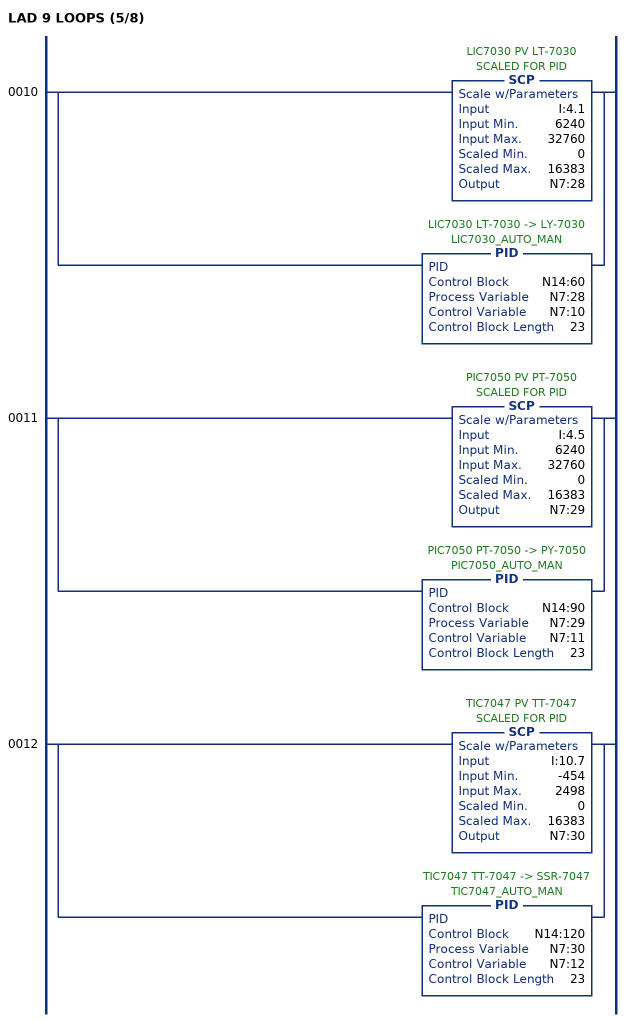
% Rung: 10 %
SOR BST SCP I:4.1 6240 32760 0 16383 N7:28 NXB PID N14:60 N7:28 N7:10 23 BND EOR
%   I:4.1  LT_7030  "LT-7030 ANALOG IN" %
%   N7:28  "LIC7030 PV LT-7030 SCALED FOR PID" %
%   N14:60  LIC7030_AUTO_MAN  "LIC7030 LT-7030 -> LY-7030" %
%   N7:10  "LY-7030 PID OP" %
% Rung: 11 %
SOR BST SCP I:4.5 6240 32760 0 16383 N7:29 NXB PID N14:90 N7:29 N7:11 23 BND EOR
%   I:4.5  PT_7050  "PT-7050 ANALOG IN" %
%   N7:29  "PIC7050 PV PT-7050 SCALED FOR PID" %
%   N14:90  PIC7050_AUTO_MAN  "PIC7050 PT-7050 -> PY-7050" %
%   N7:11  "PY-7050 PID OP" %
% Rung: 12 %
SOR BST SCP I:10.7 -454 2498 0 16383 N7:30 NXB PID N14:120 N7:30 N7:12 23 BND EOR
%   I:10.7  TT_7047  "TT-7047 ANALOG IN" %
%   N7:30  "TIC7047 PV TT-7047 SCALED FOR PID" %
%   N14:120  TIC7047_AUTO_MAN  "TIC7047 TT-7047 -> SSR-7047" %
%   N7:12  "SSR-7047 PID OP" %

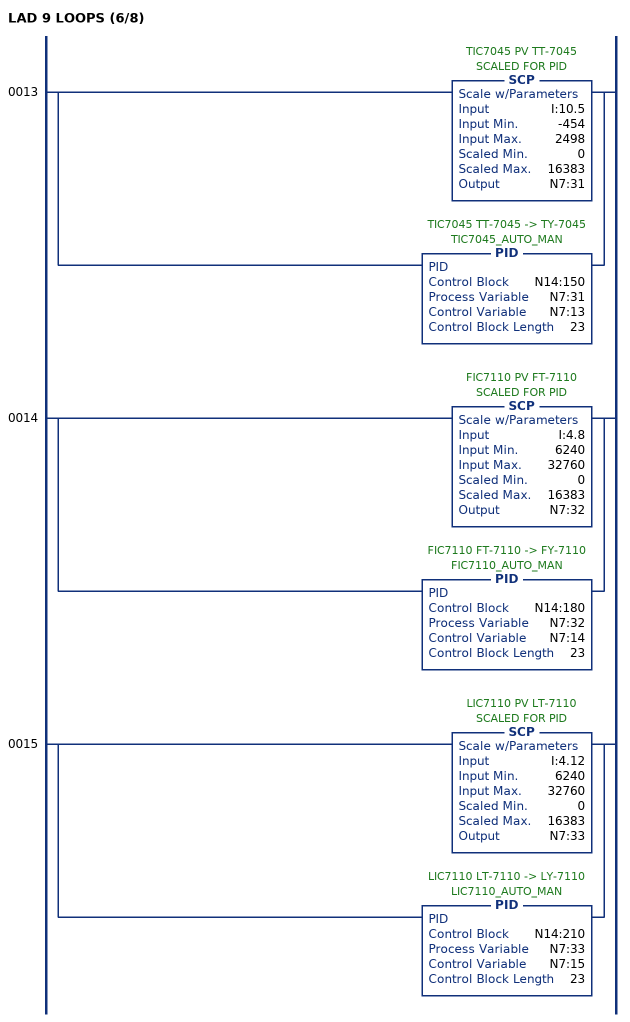
% Rung: 13 %
SOR BST SCP I:10.5 -454 2498 0 16383 N7:31 NXB PID N14:150 N7:31 N7:13 23 BND EOR
%   I:10.5  TT_7045  "TT-7045 ANALOG IN" %
%   N7:31  "TIC7045 PV TT-7045 SCALED FOR PID" %
%   N14:150  TIC7045_AUTO_MAN  "TIC7045 TT-7045 -> TY-7045" %
%   N7:13  "TY-7045 PID OP" %
% Rung: 14 %
SOR BST SCP I:4.8 6240 32760 0 16383 N7:32 NXB PID N14:180 N7:32 N7:14 23 BND EOR
%   I:4.8  FT_7110  "FT-7110 ANALOG IN" %
%   N7:32  "FIC7110 PV FT-7110 SCALED FOR PID" %
%   N14:180  FIC7110_AUTO_MAN  "FIC7110 FT-7110 -> FY-7110" %
%   N7:14  "FY-7110 PID OP" %
% Rung: 15 %
SOR BST SCP I:4.12 6240 32760 0 16383 N7:33 NXB PID N14:210 N7:33 N7:15 23 BND EOR
%   I:4.12  LT_7110  "LT-7110 ANALOG IN" %
%   N7:33  "LIC7110 PV LT-7110 SCALED FOR PID" %
%   N14:210  LIC7110_AUTO_MAN  "LIC7110 LT-7110 -> LY-7110" %
%   N7:15  "LY-7110 PID OP" %

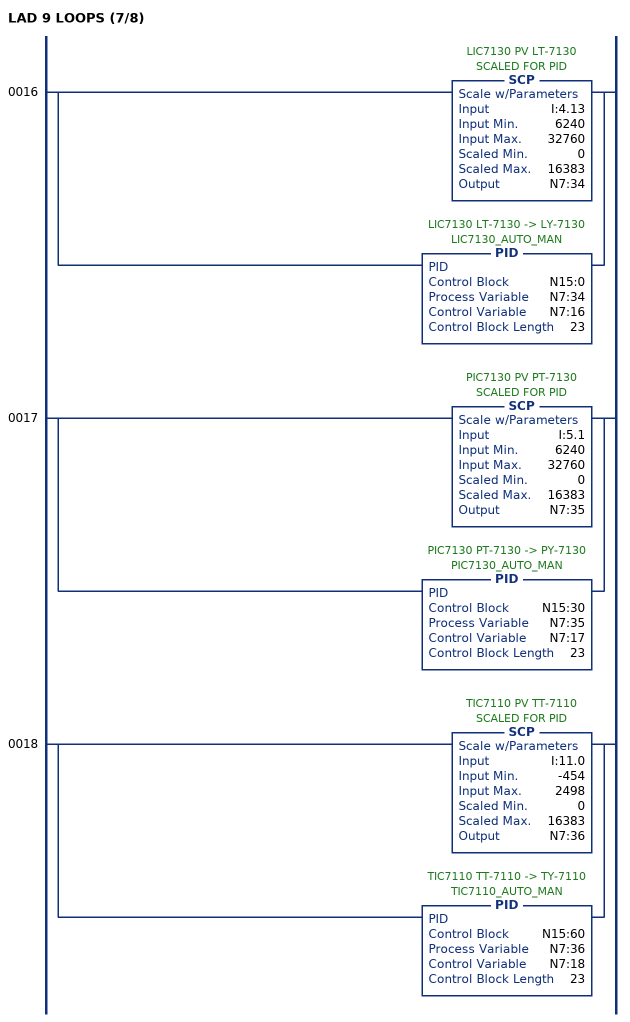
% Rung: 16 %
SOR BST SCP I:4.13 6240 32760 0 16383 N7:34 NXB PID N15:0 N7:34 N7:16 23 BND EOR
%   I:4.13  LT_7130  "LT-7130 ANALOG IN" %
%   N7:34  "LIC7130 PV LT-7130 SCALED FOR PID" %
%   N15:0  LIC7130_AUTO_MAN  "LIC7130 LT-7130 -> LY-7130" %
%   N7:16  "LY-7130 PID OP" %
% Rung: 17 %
SOR BST SCP I:5.1 6240 32760 0 16383 N7:35 NXB PID N15:30 N7:35 N7:17 23 BND EOR
%   I:5.1  PT_7130  "PT-7130 ANALOG IN" %
%   N7:35  "PIC7130 PV PT-7130 SCALED FOR PID" %
%   N15:30  PIC7130_AUTO_MAN  "PIC7130 PT-7130 -> PY-7130" %
%   N7:17  "PY-7130 PID OP" %
% Rung: 18 %
SOR BST SCP I:11.0 -454 2498 0 16383 N7:36 NXB PID N15:60 N7:36 N7:18 23 BND EOR
%   I:11.0  TT_7110  "TT-7110 ANALOG IN" %
%   N7:36  "TIC7110 PV TT-7110 SCALED FOR PID" %
%   N15:60  TIC7110_AUTO_MAN  "TIC7110 TT-7110 -> TY-7110" %
%   N7:18  "TY-7110 PID OP" %

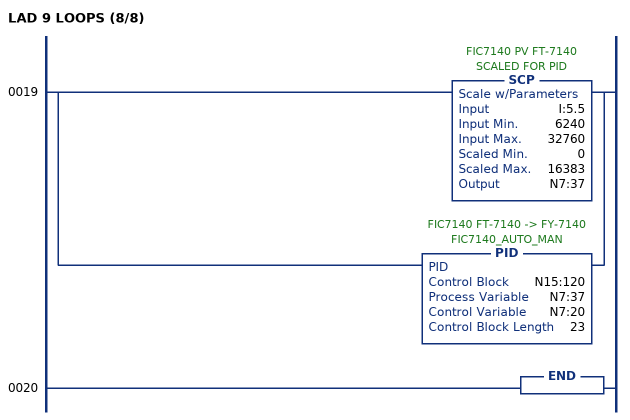
% Rung: 19 %
SOR BST SCP I:5.5 6240 32760 0 16383 N7:37 NXB PID N15:120 N7:37 N7:20 23 BND EOR
%   I:5.5  FT_7140  "FT-7140 ANALOG IN" %
%   N7:37  "FIC7140 PV FT-7140 SCALED FOR PID" %
%   N15:120  FIC7140_AUTO_MAN  "FIC7140 FT-7140 -> FY-7140" %
%   N7:20  "FY-7140 PID OP" %
% Rung: 20 %
SOR END EOR

LADDER 10 "CONTROL"
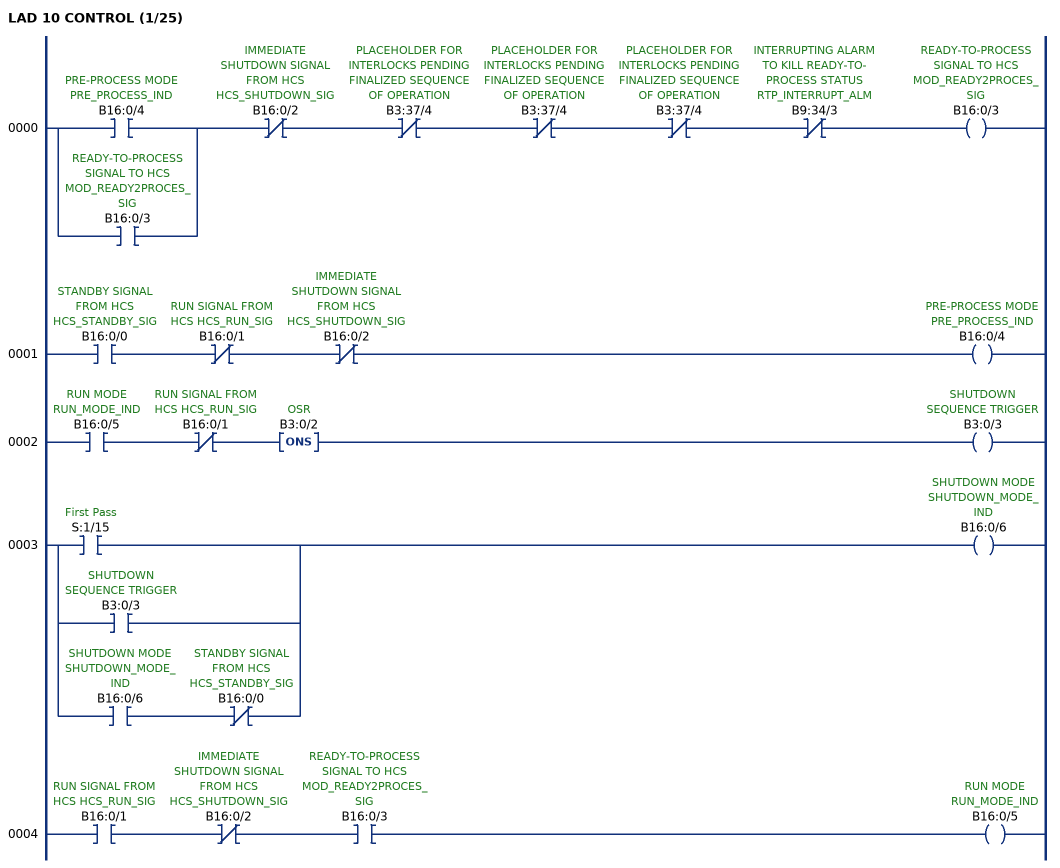
% Rung: 0 %
SOR BST XIC B16:0/4 NXB XIC B16:0/3 BND XIO B16:0/2 XIO B3:37/4 XIO B3:37/4 XIO B3:37/4 XIO B9:34/3 OTE B16:0/3 EOR
%   B16:0/4  PRE_PROCESS_IND  "PRE-PROCESS MODE" %
%   B16:0/3  MOD_READY2PROCES_SIG  "READY-TO-PROCESS SIGNAL TO HCS" %
%   B16:0/2  HCS_SHUTDOWN_SIG  "IMMEDIATE SHUTDOWN SIGNAL FROM HCS" %
%   B3:37/4  "PLACEHOLDER FOR INTERLOCKS PENDING FINALIZED SEQUENCE OF OPERATION" %
%   B9:34/3  RTP_INTERRUPT_ALM  "INTERRUPTING ALARM TO KILL READY-TO-PROCESS STATUS" %
% Rung: 1 %
SOR XIC B16:0/0 XIO B16:0/1 XIO B16:0/2 OTE B16:0/4 EOR
%   B16:0/0  HCS_STANDBY_SIG  "STANDBY SIGNAL FROM HCS" %
%   B16:0/1  HCS_RUN_SIG  "RUN SIGNAL FROM HCS" %
%   B16:0/2  HCS_SHUTDOWN_SIG  "IMMEDIATE SHUTDOWN SIGNAL FROM HCS" %
%   B16:0/4  PRE_PROCESS_IND  "PRE-PROCESS MODE" %
% Rung: 2 %
SOR XIC B16:0/5 XIO B16:0/1 OSR B3:0/2 OTE B3:0/3 EOR
%   B16:0/5  RUN_MODE_IND  "RUN MODE" %
%   B16:0/1  HCS_RUN_SIG  "RUN SIGNAL FROM HCS" %
%   B3:0/2  "OSR" %
%   B3:0/3  "SHUTDOWN SEQUENCE TRIGGER" %
% Rung: 3 %
SOR BST XIC S:1/15 NXB XIC B3:0/3 NXB XIC B16:0/6 XIO B16:0/0 BND OTE B16:0/6 EOR
%   S:1/15  "First Pass" %
%   B3:0/3  "SHUTDOWN SEQUENCE TRIGGER" %
%   B16:0/6  SHUTDOWN_MODE_IND  "SHUTDOWN MODE" %
%   B16:0/0  HCS_STANDBY_SIG  "STANDBY SIGNAL FROM HCS" %
% Rung: 4 %
SOR XIC B16:0/1 XIO B16:0/2 XIC B16:0/3 OTE B16:0/5 EOR
%   B16:0/1  HCS_RUN_SIG  "RUN SIGNAL FROM HCS" %
%   B16:0/2  HCS_SHUTDOWN_SIG  "IMMEDIATE SHUTDOWN SIGNAL FROM HCS" %
%   B16:0/3  MOD_READY2PROCES_SIG  "READY-TO-PROCESS SIGNAL TO HCS" %
%   B16:0/5  RUN_MODE_IND  "RUN MODE" %

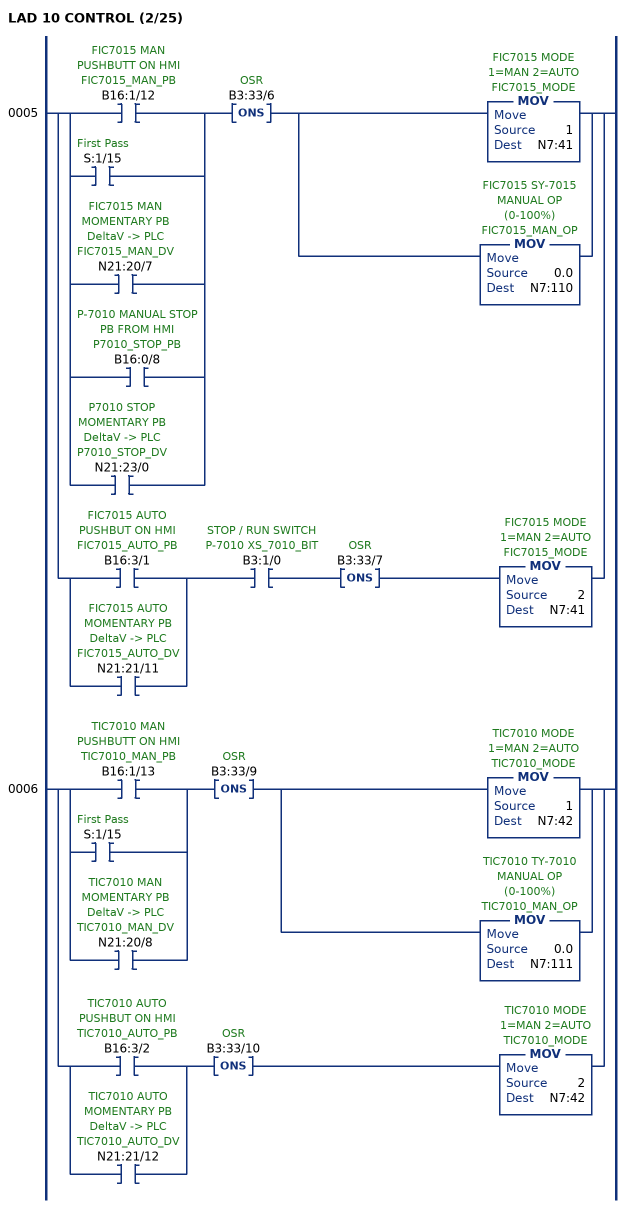
% Rung: 5 %
SOR BST BST XIC B16:1/12 NXB XIC S:1/15 NXB XIC N21:20/7 NXB XIC B16:0/8 NXB XIC N21:23/0 BND OSR B3:33/6 BST MOV 1 N7:41 NXB MOV 0.0 N7:110 BND NXB BST XIC B16:3/1 NXB XIC N21:21/11 BND XIC B3:1/0 OSR B3:33/7 MOV 2 N7:41 BND EOR
%   B16:1/12  FIC7015_MAN_PB  "FIC7015 MAN PUSHBUTT ON HMI" %
%   S:1/15  "First Pass" %
%   N21:20/7  FIC7015_MAN_DV  "FIC7015 MAN MOMENTARY PB DeltaV -> PLC" %
%   B16:0/8  P7010_STOP_PB  "P-7010 MANUAL STOP PB FROM HMI" %
%   N21:23/0  P7010_STOP_DV  "P7010 STOP MOMENTARY PB DeltaV -> PLC" %
%   B3:33/6  "OSR" %
%   N7:41  FIC7015_MODE  "FIC7015 MODE 1=MAN 2=AUTO" %
%   N7:110  FIC7015_MAN_OP  "FIC7015 SY-7015 MANUAL OP (0-100%)" %
%   B16:3/1  FIC7015_AUTO_PB  "FIC7015 AUTO PUSHBUT ON HMI" %
%   N21:21/11  FIC7015_AUTO_DV  "FIC7015 AUTO MOMENTARY PB DeltaV -> PLC" %
%   B3:1/0  XS_7010_BIT  "STOP / RUN SWITCH P-7010" %
%   B3:33/7  "OSR" %
% Rung: 6 %
SOR BST BST XIC B16:1/13 NXB XIC S:1/15 NXB XIC N21:20/8 BND OSR B3:33/9 BST MOV 1 N7:42 NXB MOV 0.0 N7:111 BND NXB BST XIC B16:3/2 NXB XIC N21:21/12 BND OSR B3:33/10 MOV 2 N7:42 BND EOR
%   B16:1/13  TIC7010_MAN_PB  "TIC7010 MAN PUSHBUTT ON HMI" %
%   S:1/15  "First Pass" %
%   N21:20/8  TIC7010_MAN_DV  "TIC7010 MAN MOMENTARY PB DeltaV -> PLC" %
%   B3:33/9  "OSR" %
%   N7:42  TIC7010_MODE  "TIC7010 MODE 1=MAN 2=AUTO" %
%   N7:111  TIC7010_MAN_OP  "TIC7010 TY-7010 MANUAL OP (0-100%)" %
%   B16:3/2  TIC7010_AUTO_PB  "TIC7010 AUTO PUSHBUT ON HMI" %
%   N21:21/12  TIC7010_AUTO_DV  "TIC7010 AUTO MOMENTARY PB DeltaV -> PLC" %
%   B3:33/10  "OSR" %

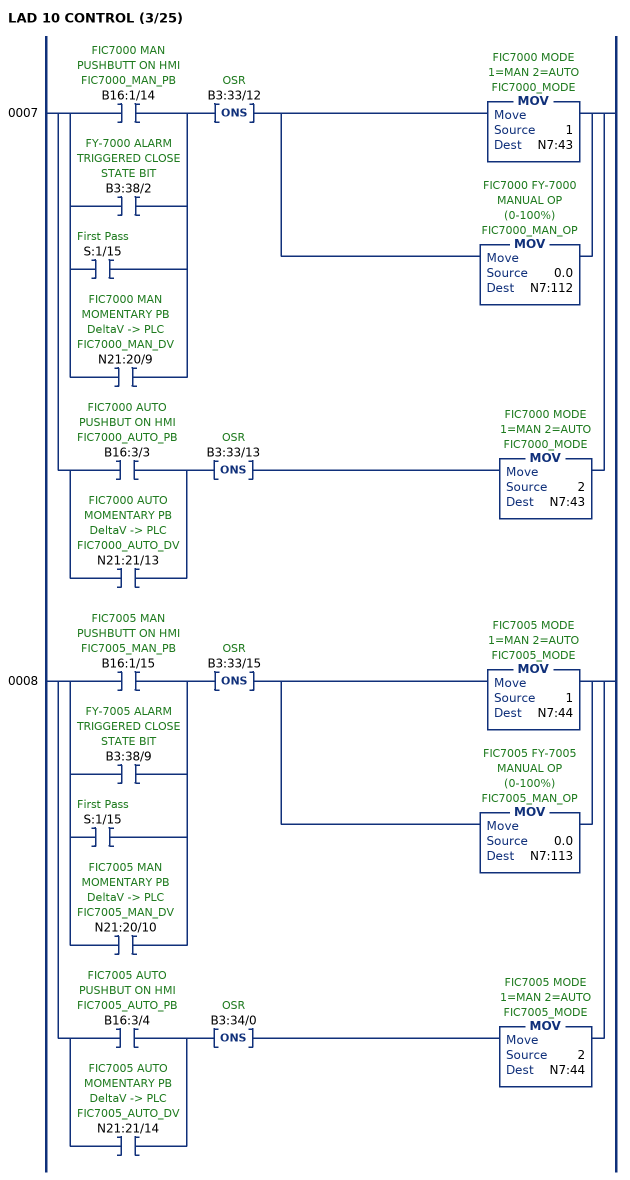
% Rung: 7 %
SOR BST BST XIC B16:1/14 NXB XIC B3:38/2 NXB XIC S:1/15 NXB XIC N21:20/9 BND OSR B3:33/12 BST MOV 1 N7:43 NXB MOV 0.0 N7:112 BND NXB BST XIC B16:3/3 NXB XIC N21:21/13 BND OSR B3:33/13 MOV 2 N7:43 BND EOR
%   B16:1/14  FIC7000_MAN_PB  "FIC7000 MAN PUSHBUTT ON HMI" %
%   B3:38/2  "FY-7000 ALARM TRIGGERED CLOSE STATE BIT" %
%   S:1/15  "First Pass" %
%   N21:20/9  FIC7000_MAN_DV  "FIC7000 MAN MOMENTARY PB DeltaV -> PLC" %
%   B3:33/12  "OSR" %
%   N7:43  FIC7000_MODE  "FIC7000 MODE 1=MAN 2=AUTO" %
%   N7:112  FIC7000_MAN_OP  "FIC7000 FY-7000 MANUAL OP (0-100%)" %
%   B16:3/3  FIC7000_AUTO_PB  "FIC7000 AUTO PUSHBUT ON HMI" %
%   N21:21/13  FIC7000_AUTO_DV  "FIC7000 AUTO MOMENTARY PB DeltaV -> PLC" %
%   B3:33/13  "OSR" %
% Rung: 8 %
SOR BST BST XIC B16:1/15 NXB XIC B3:38/9 NXB XIC S:1/15 NXB XIC N21:20/10 BND OSR B3:33/15 BST MOV 1 N7:44 NXB MOV 0.0 N7:113 BND NXB BST XIC B16:3/4 NXB XIC N21:21/14 BND OSR B3:34/0 MOV 2 N7:44 BND EOR
%   B16:1/15  FIC7005_MAN_PB  "FIC7005 MAN PUSHBUTT ON HMI" %
%   B3:38/9  "FY-7005 ALARM TRIGGERED CLOSE STATE BIT" %
%   S:1/15  "First Pass" %
%   N21:20/10  FIC7005_MAN_DV  "FIC7005 MAN MOMENTARY PB DeltaV -> PLC" %
%   B3:33/15  "OSR" %
%   N7:44  FIC7005_MODE  "FIC7005 MODE 1=MAN 2=AUTO" %
%   N7:113  FIC7005_MAN_OP  "FIC7005 FY-7005 MANUAL OP (0-100%)" %
%   B16:3/4  FIC7005_AUTO_PB  "FIC7005 AUTO PUSHBUT ON HMI" %
%   N21:21/14  FIC7005_AUTO_DV  "FIC7005 AUTO MOMENTARY PB DeltaV -> PLC" %
%   B3:34/0  "OSR" %

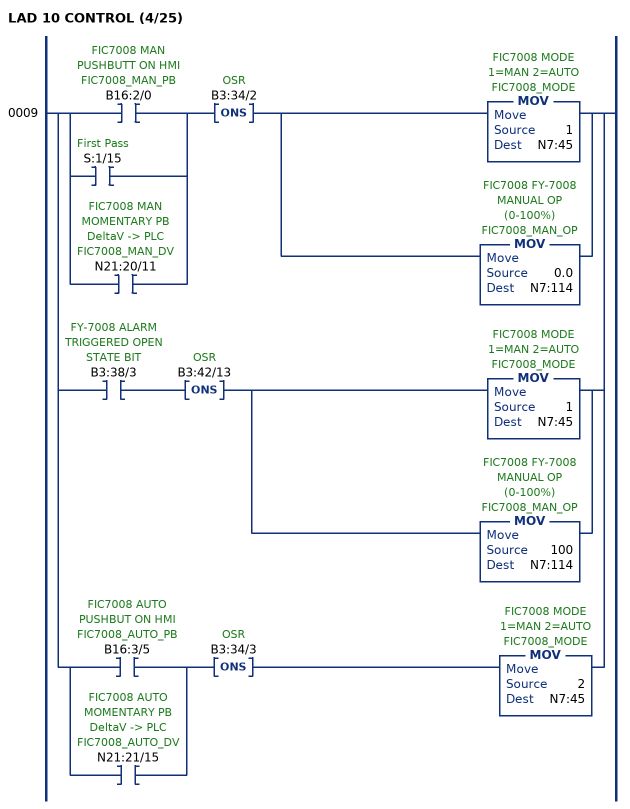
% Rung: 9 %
SOR BST BST XIC B16:2/0 NXB XIC S:1/15 NXB XIC N21:20/11 BND OSR B3:34/2 BST MOV 1 N7:45 NXB MOV 0.0 N7:114 BND NXB XIC B3:38/3 OSR B3:42/13 BST MOV 1 N7:45 NXB MOV 100 N7:114 BND NXB BST XIC B16:3/5 NXB XIC N21:21/15 BND OSR B3:34/3 MOV 2 N7:45 BND EOR
%   B16:2/0  FIC7008_MAN_PB  "FIC7008 MAN PUSHBUTT ON HMI" %
%   S:1/15  "First Pass" %
%   N21:20/11  FIC7008_MAN_DV  "FIC7008 MAN MOMENTARY PB DeltaV -> PLC" %
%   B3:34/2  "OSR" %
%   N7:45  FIC7008_MODE  "FIC7008 MODE 1=MAN 2=AUTO" %
%   N7:114  FIC7008_MAN_OP  "FIC7008 FY-7008 MANUAL OP (0-100%)" %
%   B3:38/3  "FY-7008 ALARM TRIGGERED OPEN STATE BIT" %
%   B3:42/13  "OSR" %
%   B16:3/5  FIC7008_AUTO_PB  "FIC7008 AUTO PUSHBUT ON HMI" %
%   N21:21/15  FIC7008_AUTO_DV  "FIC7008 AUTO MOMENTARY PB DeltaV -> PLC" %
%   B3:34/3  "OSR" %

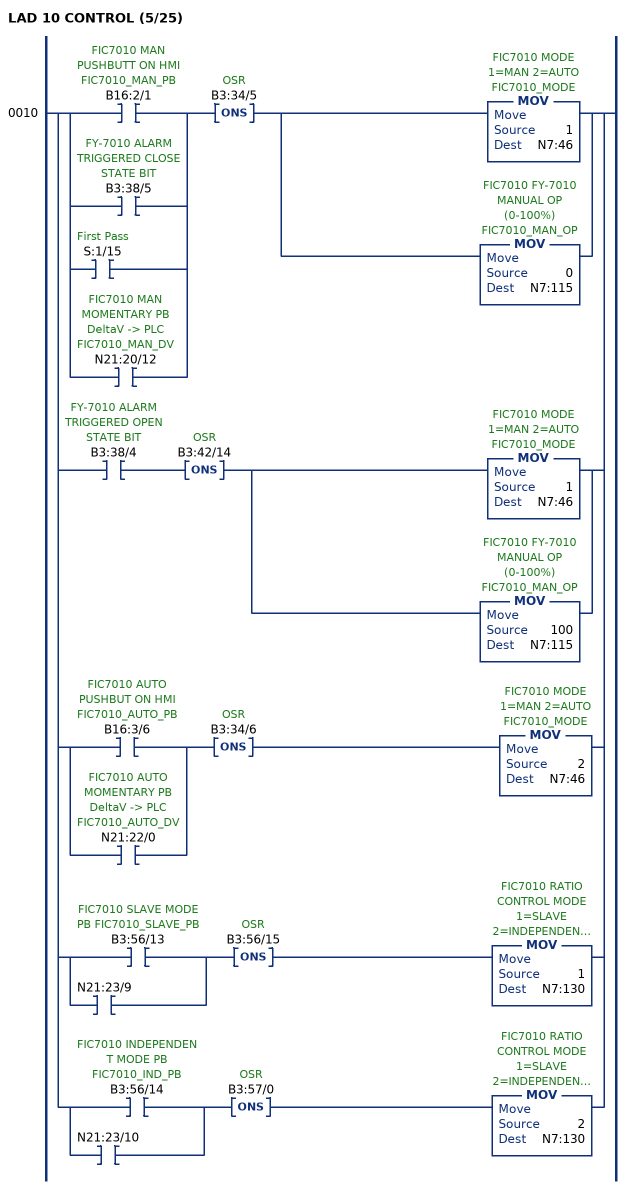
% Rung: 10 %
SOR BST BST XIC B16:2/1 NXB XIC B3:38/5 NXB XIC S:1/15 NXB XIC N21:20/12 BND OSR B3:34/5 BST MOV 1 N7:46 NXB MOV 0 N7:115 BND NXB XIC B3:38/4 OSR B3:42/14 BST MOV 1 N7:46 NXB MOV 100 N7:115 BND NXB BST XIC B16:3/6 NXB XIC N21:22/0 BND OSR B3:34/6 MOV 2 N7:46 NXB BST XIC B3:56/13 NXB XIC N21:23/9 BND OSR B3:56/15 MOV 1 N7:130 NXB BST XIC B3:56/14 NXB XIC N21:23/10 BND OSR B3:57/0 MOV 2 N7:130 BND EOR
%   B16:2/1  FIC7010_MAN_PB  "FIC7010 MAN PUSHBUTT ON HMI" %
%   B3:38/5  "FY-7010 ALARM TRIGGERED CLOSE STATE BIT" %
%   S:1/15  "First Pass" %
%   N21:20/12  FIC7010_MAN_DV  "FIC7010 MAN MOMENTARY PB DeltaV -> PLC" %
%   B3:34/5  "OSR" %
%   N7:46  FIC7010_MODE  "FIC7010 MODE 1=MAN 2=AUTO" %
%   N7:115  FIC7010_MAN_OP  "FIC7010 FY-7010 MANUAL OP (0-100%)" %
%   B3:38/4  "FY-7010 ALARM TRIGGERED OPEN STATE BIT" %
%   B3:42/14  "OSR" %
%   B16:3/6  FIC7010_AUTO_PB  "FIC7010 AUTO PUSHBUT ON HMI" %
%   N21:22/0  FIC7010_AUTO_DV  "FIC7010 AUTO MOMENTARY PB DeltaV -> PLC" %
%   B3:34/6  "OSR" %
%   B3:56/13  FIC7010_SLAVE_PB  "FIC7010 SLAVE MODE PB" %
%   B3:56/15  "OSR" %
%   N7:130  FIC7010_RATIO_MODE  "FIC7010 RATIO CONTROL MODE 1=SLAVE 2=INDEPENDENT" %
%   B3:56/14  FIC7010_IND_PB  "FIC7010 INDEPENDENT MODE PB" %
%   B3:57/0  "OSR" %

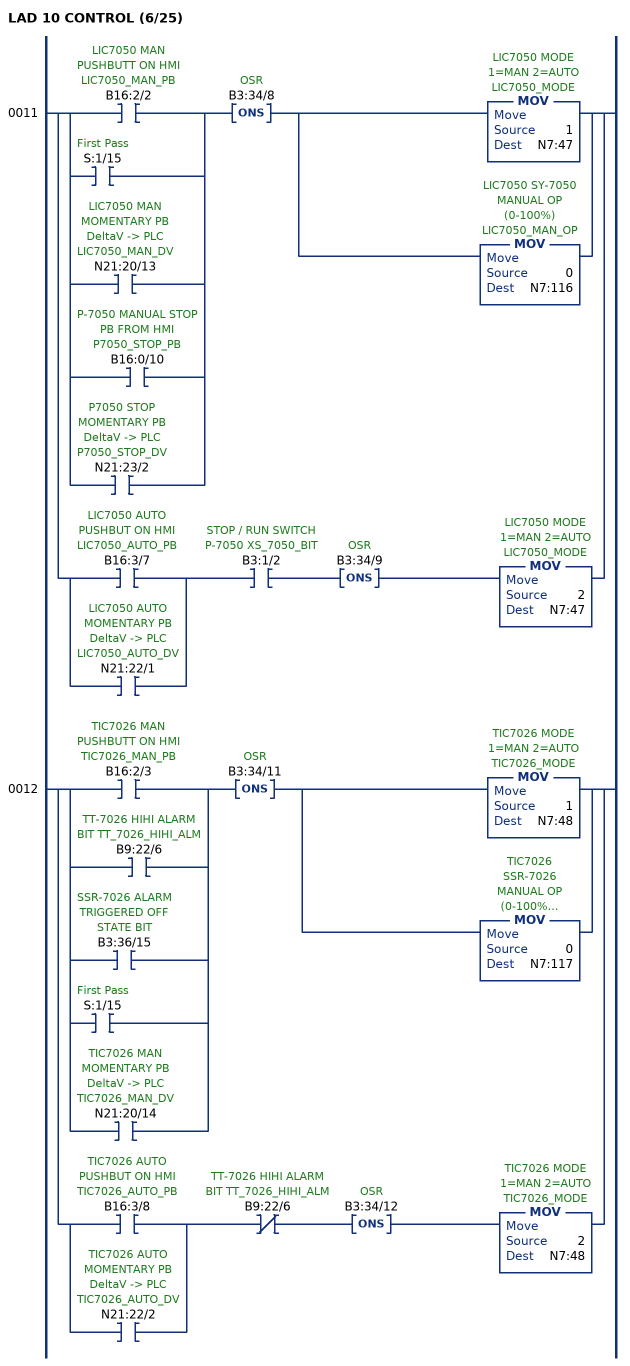
% Rung: 11 %
SOR BST BST XIC B16:2/2 NXB XIC S:1/15 NXB XIC N21:20/13 NXB XIC B16:0/10 NXB XIC N21:23/2 BND OSR B3:34/8 BST MOV 1 N7:47 NXB MOV 0 N7:116 BND NXB BST XIC B16:3/7 NXB XIC N21:22/1 BND XIC B3:1/2 OSR B3:34/9 MOV 2 N7:47 BND EOR
%   B16:2/2  LIC7050_MAN_PB  "LIC7050 MAN PUSHBUTT ON HMI" %
%   S:1/15  "First Pass" %
%   N21:20/13  LIC7050_MAN_DV  "LIC7050 MAN MOMENTARY PB DeltaV -> PLC" %
%   B16:0/10  P7050_STOP_PB  "P-7050 MANUAL STOP PB FROM HMI" %
%   N21:23/2  P7050_STOP_DV  "P7050 STOP MOMENTARY PB DeltaV -> PLC" %
%   B3:34/8  "OSR" %
%   N7:47  LIC7050_MODE  "LIC7050 MODE 1=MAN 2=AUTO" %
%   N7:116  LIC7050_MAN_OP  "LIC7050 SY-7050 MANUAL OP (0-100%)" %
%   B16:3/7  LIC7050_AUTO_PB  "LIC7050 AUTO PUSHBUT ON HMI" %
%   N21:22/1  LIC7050_AUTO_DV  "LIC7050 AUTO MOMENTARY PB DeltaV -> PLC" %
%   B3:1/2  XS_7050_BIT  "STOP / RUN SWITCH P-7050" %
%   B3:34/9  "OSR" %
% Rung: 12 %
SOR BST BST XIC B16:2/3 NXB XIC B9:22/6 NXB XIC B3:36/15 NXB XIC S:1/15 NXB XIC N21:20/14 BND OSR B3:34/11 BST MOV 1 N7:48 NXB MOV 0 N7:117 BND NXB BST XIC B16:3/8 NXB XIC N21:22/2 BND XIO B9:22/6 OSR B3:34/12 MOV 2 N7:48 BND EOR
%   B16:2/3  TIC7026_MAN_PB  "TIC7026 MAN PUSHBUTT ON HMI" %
%   B9:22/6  TT_7026_HIHI_ALM  "TT-7026 HIHI ALARM BIT" %
%   B3:36/15  "SSR-7026 ALARM TRIGGERED OFF STATE BIT" %
%   S:1/15  "First Pass" %
%   N21:20/14  TIC7026_MAN_DV  "TIC7026 MAN MOMENTARY PB DeltaV -> PLC" %
%   B3:34/11  "OSR" %
%   N7:48  TIC7026_MODE  "TIC7026 MODE 1=MAN 2=AUTO" %
%   N7:117  TIC7026_MAN_OP  "TIC7026 SSR-7026 MANUAL OP (0-100%)" %
%   B16:3/8  TIC7026_AUTO_PB  "TIC7026 AUTO PUSHBUT ON HMI" %
%   N21:22/2  TIC7026_AUTO_DV  "TIC7026 AUTO MOMENTARY PB DeltaV -> PLC" %
%   B3:34/12  "OSR" %

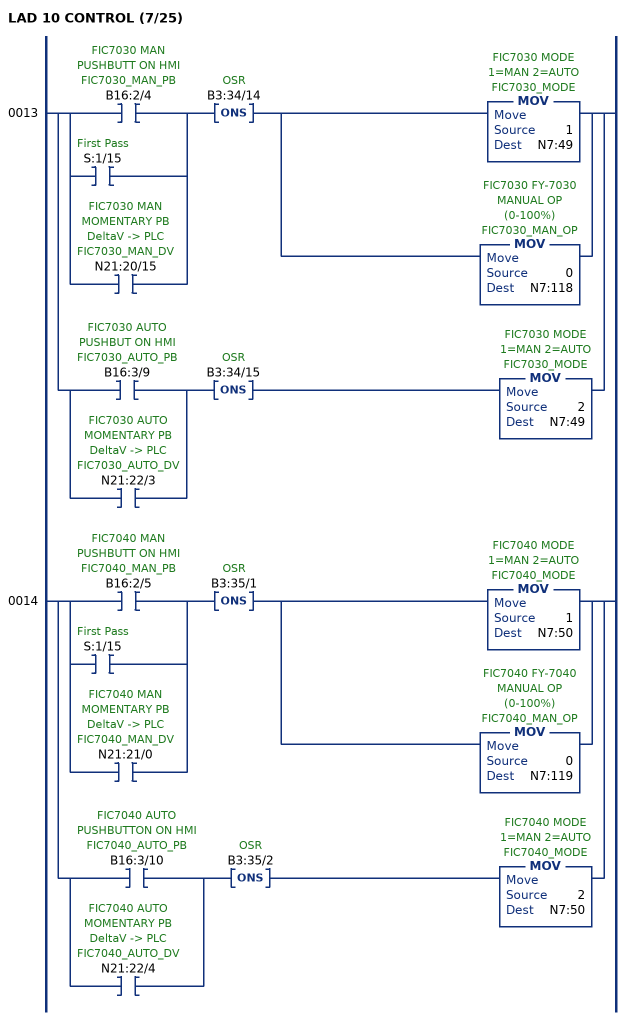
% Rung: 13 %
SOR BST BST XIC B16:2/4 NXB XIC S:1/15 NXB XIC N21:20/15 BND OSR B3:34/14 BST MOV 1 N7:49 NXB MOV 0 N7:118 BND NXB BST XIC B16:3/9 NXB XIC N21:22/3 BND OSR B3:34/15 MOV 2 N7:49 BND EOR
%   B16:2/4  FIC7030_MAN_PB  "FIC7030 MAN PUSHBUTT ON HMI" %
%   S:1/15  "First Pass" %
%   N21:20/15  FIC7030_MAN_DV  "FIC7030 MAN MOMENTARY PB DeltaV -> PLC" %
%   B3:34/14  "OSR" %
%   N7:49  FIC7030_MODE  "FIC7030 MODE 1=MAN 2=AUTO" %
%   N7:118  FIC7030_MAN_OP  "FIC7030 FY-7030 MANUAL OP (0-100%)" %
%   B16:3/9  FIC7030_AUTO_PB  "FIC7030 AUTO PUSHBUT ON HMI" %
%   N21:22/3  FIC7030_AUTO_DV  "FIC7030 AUTO MOMENTARY PB DeltaV -> PLC" %
%   B3:34/15  "OSR" %
% Rung: 14 %
SOR BST BST XIC B16:2/5 NXB XIC S:1/15 NXB XIC N21:21/0 BND OSR B3:35/1 BST MOV 1 N7:50 NXB MOV 0 N7:119 BND NXB BST XIC B16:3/10 NXB XIC N21:22/4 BND OSR B3:35/2 MOV 2 N7:50 BND EOR
%   B16:2/5  FIC7040_MAN_PB  "FIC7040 MAN PUSHBUTT ON HMI" %
%   S:1/15  "First Pass" %
%   N21:21/0  FIC7040_MAN_DV  "FIC7040 MAN MOMENTARY PB DeltaV -> PLC" %
%   B3:35/1  "OSR" %
%   N7:50  FIC7040_MODE  "FIC7040 MODE 1=MAN 2=AUTO" %
%   N7:119  FIC7040_MAN_OP  "FIC7040 FY-7040 MANUAL OP (0-100%)" %
%   B16:3/10  FIC7040_AUTO_PB  "FIC7040 AUTO PUSHBUTTON ON HMI" %
%   N21:22/4  FIC7040_AUTO_DV  "FIC7040 AUTO MOMENTARY PB DeltaV -> PLC" %
%   B3:35/2  "OSR" %

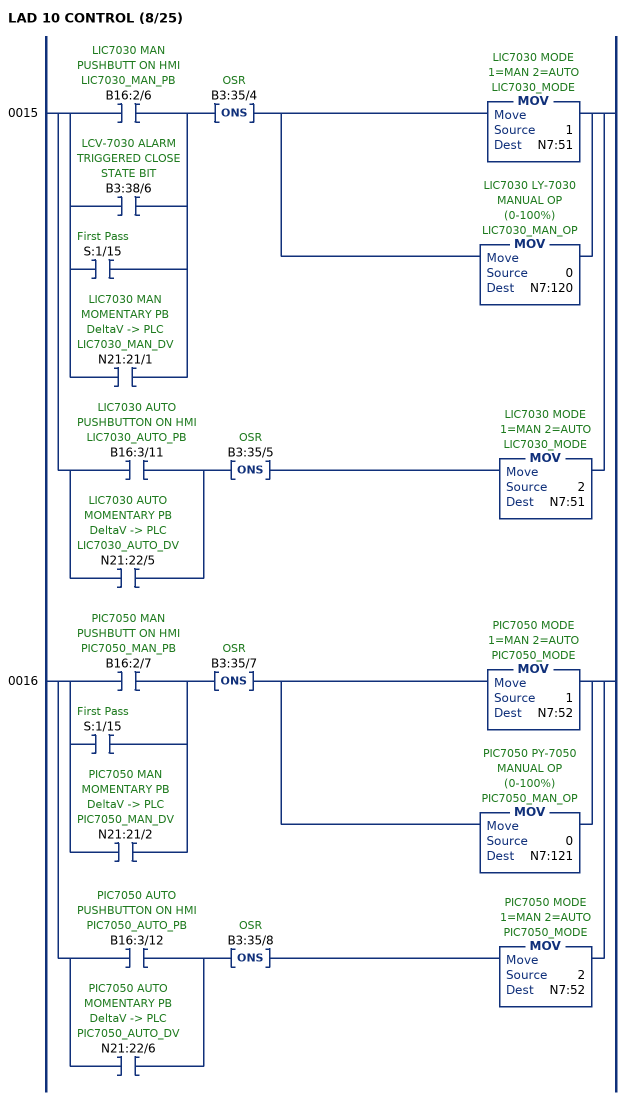
% Rung: 15 %
SOR BST BST XIC B16:2/6 NXB XIC B3:38/6 NXB XIC S:1/15 NXB XIC N21:21/1 BND OSR B3:35/4 BST MOV 1 N7:51 NXB MOV 0 N7:120 BND NXB BST XIC B16:3/11 NXB XIC N21:22/5 BND OSR B3:35/5 MOV 2 N7:51 BND EOR
%   B16:2/6  LIC7030_MAN_PB  "LIC7030 MAN PUSHBUTT ON HMI" %
%   B3:38/6  "LCV-7030 ALARM TRIGGERED CLOSE STATE BIT" %
%   S:1/15  "First Pass" %
%   N21:21/1  LIC7030_MAN_DV  "LIC7030 MAN MOMENTARY PB DeltaV -> PLC" %
%   B3:35/4  "OSR" %
%   N7:51  LIC7030_MODE  "LIC7030 MODE 1=MAN 2=AUTO" %
%   N7:120  LIC7030_MAN_OP  "LIC7030 LY-7030 MANUAL OP (0-100%)" %
%   B16:3/11  LIC7030_AUTO_PB  "LIC7030 AUTO PUSHBUTTON ON HMI" %
%   N21:22/5  LIC7030_AUTO_DV  "LIC7030 AUTO MOMENTARY PB DeltaV -> PLC" %
%   B3:35/5  "OSR" %
% Rung: 16 %
SOR BST BST XIC B16:2/7 NXB XIC S:1/15 NXB XIC N21:21/2 BND OSR B3:35/7 BST MOV 1 N7:52 NXB MOV 0 N7:121 BND NXB BST XIC B16:3/12 NXB XIC N21:22/6 BND OSR B3:35/8 MOV 2 N7:52 BND EOR
%   B16:2/7  PIC7050_MAN_PB  "PIC7050 MAN PUSHBUTT ON HMI" %
%   S:1/15  "First Pass" %
%   N21:21/2  PIC7050_MAN_DV  "PIC7050 MAN MOMENTARY PB DeltaV -> PLC" %
%   B3:35/7  "OSR" %
%   N7:52  PIC7050_MODE  "PIC7050 MODE 1=MAN 2=AUTO" %
%   N7:121  PIC7050_MAN_OP  "PIC7050 PY-7050 MANUAL OP (0-100%)" %
%   B16:3/12  PIC7050_AUTO_PB  "PIC7050 AUTO PUSHBUTTON ON HMI" %
%   N21:22/6  PIC7050_AUTO_DV  "PIC7050 AUTO MOMENTARY PB DeltaV -> PLC" %
%   B3:35/8  "OSR" %

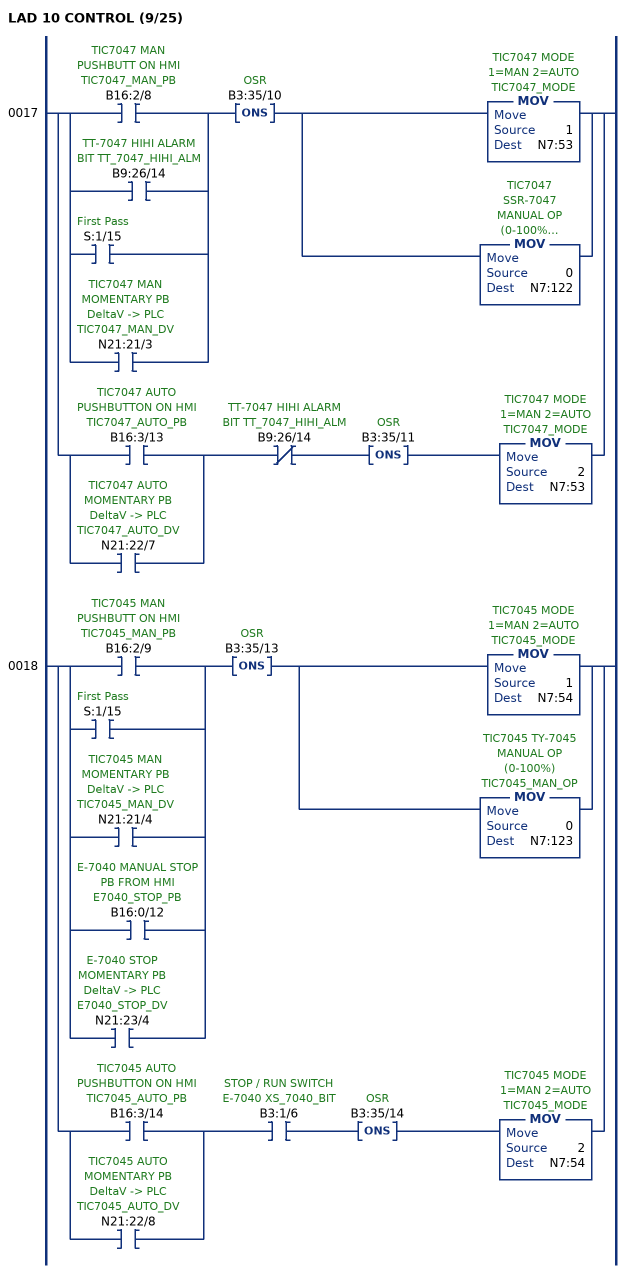
% Rung: 17 %
SOR BST BST XIC B16:2/8 NXB XIC B9:26/14 NXB XIC S:1/15 NXB XIC N21:21/3 BND OSR B3:35/10 BST MOV 1 N7:53 NXB MOV 0 N7:122 BND NXB BST XIC B16:3/13 NXB XIC N21:22/7 BND XIO B9:26/14 OSR B3:35/11 MOV 2 N7:53 BND EOR
%   B16:2/8  TIC7047_MAN_PB  "TIC7047 MAN PUSHBUTT ON HMI" %
%   B9:26/14  TT_7047_HIHI_ALM  "TT-7047 HIHI ALARM BIT" %
%   S:1/15  "First Pass" %
%   N21:21/3  TIC7047_MAN_DV  "TIC7047 MAN MOMENTARY PB DeltaV -> PLC" %
%   B3:35/10  "OSR" %
%   N7:53  TIC7047_MODE  "TIC7047 MODE 1=MAN 2=AUTO" %
%   N7:122  TIC7047_MAN_OP  "TIC7047 SSR-7047 MANUAL OP (0-100%)" %
%   B16:3/13  TIC7047_AUTO_PB  "TIC7047 AUTO PUSHBUTTON ON HMI" %
%   N21:22/7  TIC7047_AUTO_DV  "TIC7047 AUTO MOMENTARY PB DeltaV -> PLC" %
%   B3:35/11  "OSR" %
% Rung: 18 %
SOR BST BST XIC B16:2/9 NXB XIC S:1/15 NXB XIC N21:21/4 NXB XIC B16:0/12 NXB XIC N21:23/4 BND OSR B3:35/13 BST MOV 1 N7:54 NXB MOV 0 N7:123 BND NXB BST XIC B16:3/14 NXB XIC N21:22/8 BND XIC B3:1/6 OSR B3:35/14 MOV 2 N7:54 BND EOR
%   B16:2/9  TIC7045_MAN_PB  "TIC7045 MAN PUSHBUTT ON HMI" %
%   S:1/15  "First Pass" %
%   N21:21/4  TIC7045_MAN_DV  "TIC7045 MAN MOMENTARY PB DeltaV -> PLC" %
%   B16:0/12  E7040_STOP_PB  "E-7040 MANUAL STOP PB FROM HMI" %
%   N21:23/4  E7040_STOP_DV  "E-7040 STOP MOMENTARY PB DeltaV -> PLC" %
%   B3:35/13  "OSR" %
%   N7:54  TIC7045_MODE  "TIC7045 MODE 1=MAN 2=AUTO" %
%   N7:123  TIC7045_MAN_OP  "TIC7045 TY-7045 MANUAL OP (0-100%)" %
%   B16:3/14  TIC7045_AUTO_PB  "TIC7045 AUTO PUSHBUTTON ON HMI" %
%   N21:22/8  TIC7045_AUTO_DV  "TIC7045 AUTO MOMENTARY PB DeltaV -> PLC" %
%   B3:1/6  XS_7040_BIT  "STOP / RUN SWITCH E-7040" %
%   B3:35/14  "OSR" %

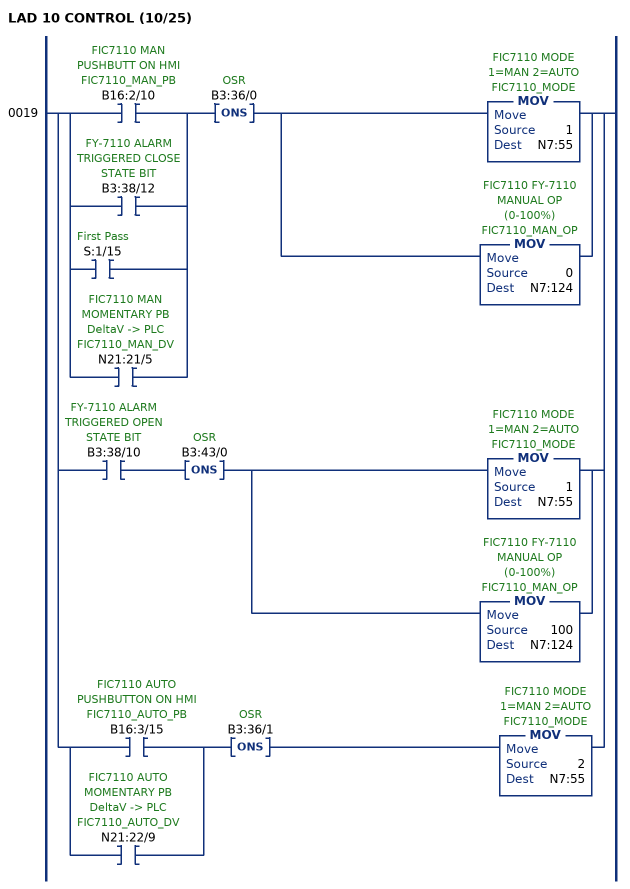
% Rung: 19 %
SOR BST BST XIC B16:2/10 NXB XIC B3:38/12 NXB XIC S:1/15 NXB XIC N21:21/5 BND OSR B3:36/0 BST MOV 1 N7:55 NXB MOV 0 N7:124 BND NXB XIC B3:38/10 OSR B3:43/0 BST MOV 1 N7:55 NXB MOV 100 N7:124 BND NXB BST XIC B16:3/15 NXB XIC N21:22/9 BND OSR B3:36/1 MOV 2 N7:55 BND EOR
%   B16:2/10  FIC7110_MAN_PB  "FIC7110 MAN PUSHBUTT ON HMI" %
%   B3:38/12  "FY-7110 ALARM TRIGGERED CLOSE STATE BIT" %
%   S:1/15  "First Pass" %
%   N21:21/5  FIC7110_MAN_DV  "FIC7110 MAN MOMENTARY PB DeltaV -> PLC" %
%   B3:36/0  "OSR" %
%   N7:55  FIC7110_MODE  "FIC7110 MODE 1=MAN 2=AUTO" %
%   N7:124  FIC7110_MAN_OP  "FIC7110 FY-7110 MANUAL OP (0-100%)" %
%   B3:38/10  "FY-7110 ALARM TRIGGERED OPEN STATE BIT" %
%   B3:43/0  "OSR" %
%   B16:3/15  FIC7110_AUTO_PB  "FIC7110 AUTO PUSHBUTTON ON HMI" %
%   N21:22/9  FIC7110_AUTO_DV  "FIC7110 AUTO MOMENTARY PB DeltaV -> PLC" %
%   B3:36/1  "OSR" %

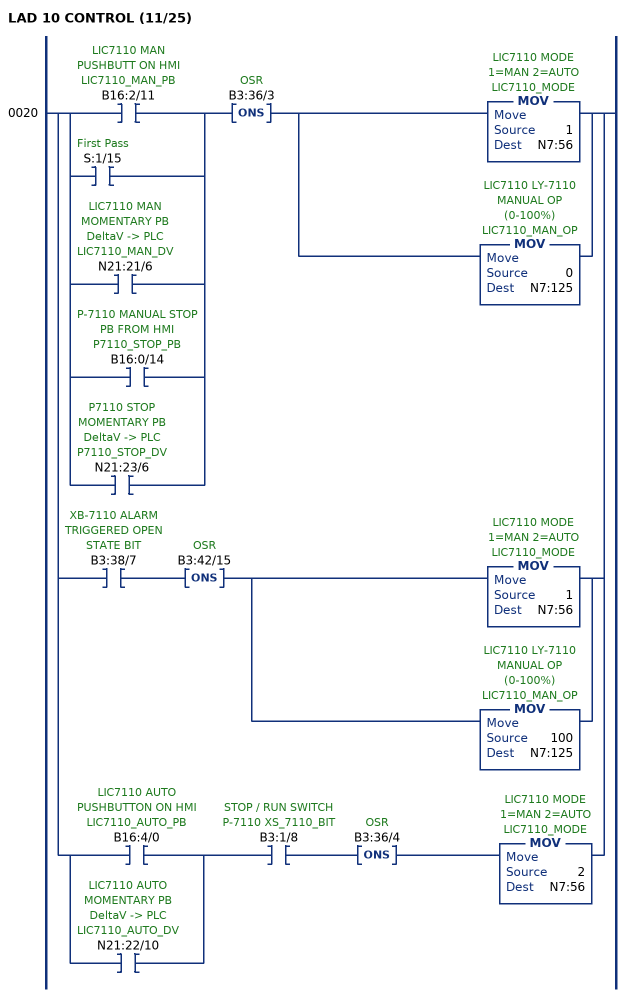
% Rung: 20 %
SOR BST BST XIC B16:2/11 NXB XIC S:1/15 NXB XIC N21:21/6 NXB XIC B16:0/14 NXB XIC N21:23/6 BND OSR B3:36/3 BST MOV 1 N7:56 NXB MOV 0 N7:125 BND NXB XIC B3:38/7 OSR B3:42/15 BST MOV 1 N7:56 NXB MOV 100 N7:125 BND NXB BST XIC B16:4/0 NXB XIC N21:22/10 BND XIC B3:1/8 OSR B3:36/4 MOV 2 N7:56 BND EOR
%   B16:2/11  LIC7110_MAN_PB  "LIC7110 MAN PUSHBUTT ON HMI" %
%   S:1/15  "First Pass" %
%   N21:21/6  LIC7110_MAN_DV  "LIC7110 MAN MOMENTARY PB DeltaV -> PLC" %
%   B16:0/14  P7110_STOP_PB  "P-7110 MANUAL STOP PB FROM HMI" %
%   N21:23/6  P7110_STOP_DV  "P7110 STOP MOMENTARY PB DeltaV -> PLC" %
%   B3:36/3  "OSR" %
%   N7:56  LIC7110_MODE  "LIC7110 MODE 1=MAN 2=AUTO" %
%   N7:125  LIC7110_MAN_OP  "LIC7110 LY-7110 MANUAL OP (0-100%)" %
%   B3:38/7  "XB-7110 ALARM TRIGGERED OPEN STATE BIT" %
%   B3:42/15  "OSR" %
%   B16:4/0  LIC7110_AUTO_PB  "LIC7110 AUTO PUSHBUTTON ON HMI" %
%   N21:22/10  LIC7110_AUTO_DV  "LIC7110 AUTO MOMENTARY PB DeltaV -> PLC" %
%   B3:1/8  XS_7110_BIT  "STOP / RUN SWITCH P-7110" %
%   B3:36/4  "OSR" %

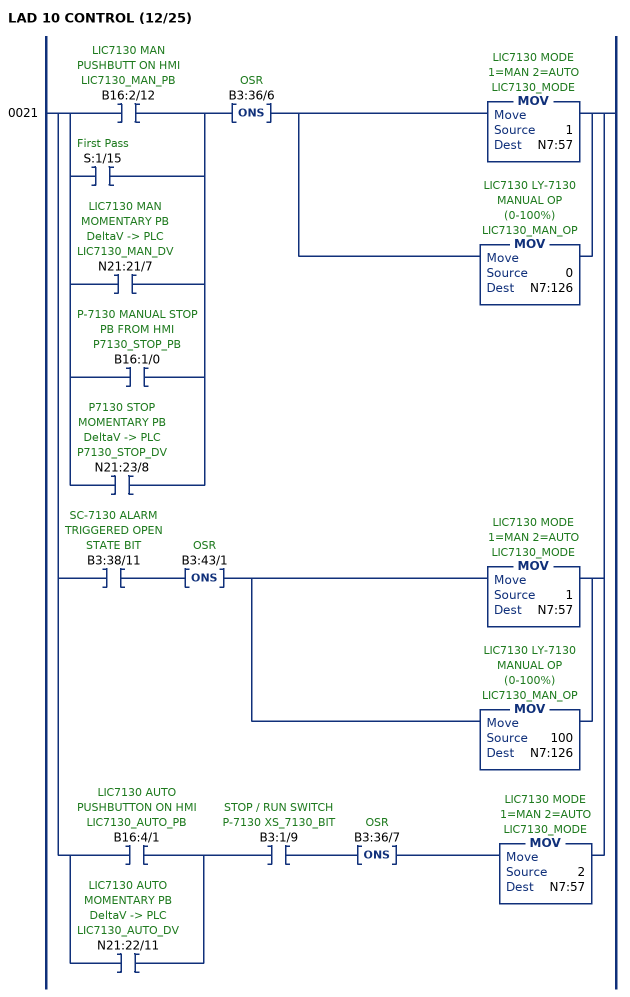
% Rung: 21 %
SOR BST BST XIC B16:2/12 NXB XIC S:1/15 NXB XIC N21:21/7 NXB XIC B16:1/0 NXB XIC N21:23/8 BND OSR B3:36/6 BST MOV 1 N7:57 NXB MOV 0 N7:126 BND NXB XIC B3:38/11 OSR B3:43/1 BST MOV 1 N7:57 NXB MOV 100 N7:126 BND NXB BST XIC B16:4/1 NXB XIC N21:22/11 BND XIC B3:1/9 OSR B3:36/7 MOV 2 N7:57 BND EOR
%   B16:2/12  LIC7130_MAN_PB  "LIC7130 MAN PUSHBUTT ON HMI" %
%   S:1/15  "First Pass" %
%   N21:21/7  LIC7130_MAN_DV  "LIC7130 MAN MOMENTARY PB DeltaV -> PLC" %
%   B16:1/0  P7130_STOP_PB  "P-7130 MANUAL STOP PB FROM HMI" %
%   N21:23/8  P7130_STOP_DV  "P7130 STOP MOMENTARY PB DeltaV -> PLC" %
%   B3:36/6  "OSR" %
%   N7:57  LIC7130_MODE  "LIC7130 MODE 1=MAN 2=AUTO" %
%   N7:126  LIC7130_MAN_OP  "LIC7130 LY-7130 MANUAL OP (0-100%)" %
%   B3:38/11  "SC-7130 ALARM TRIGGERED OPEN STATE BIT" %
%   B3:43/1  "OSR" %
%   B16:4/1  LIC7130_AUTO_PB  "LIC7130 AUTO PUSHBUTTON ON HMI" %
%   N21:22/11  LIC7130_AUTO_DV  "LIC7130 AUTO MOMENTARY PB DeltaV -> PLC" %
%   B3:1/9  XS_7130_BIT  "STOP / RUN SWITCH P-7130" %
%   B3:36/7  "OSR" %

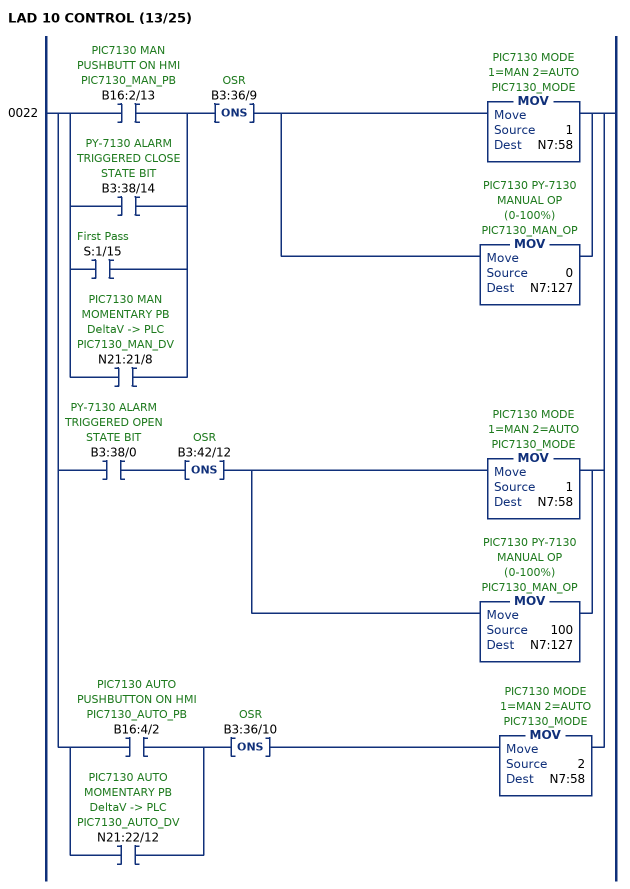
% Rung: 22 %
SOR BST BST XIC B16:2/13 NXB XIC B3:38/14 NXB XIC S:1/15 NXB XIC N21:21/8 BND OSR B3:36/9 BST MOV 1 N7:58 NXB MOV 0 N7:127 BND NXB XIC B3:38/0 OSR B3:42/12 BST MOV 1 N7:58 NXB MOV 100 N7:127 BND NXB BST XIC B16:4/2 NXB XIC N21:22/12 BND OSR B3:36/10 MOV 2 N7:58 BND EOR
%   B16:2/13  PIC7130_MAN_PB  "PIC7130 MAN PUSHBUTT ON HMI" %
%   B3:38/14  "PY-7130 ALARM TRIGGERED CLOSE STATE BIT" %
%   S:1/15  "First Pass" %
%   N21:21/8  PIC7130_MAN_DV  "PIC7130 MAN MOMENTARY PB DeltaV -> PLC" %
%   B3:36/9  "OSR" %
%   N7:58  PIC7130_MODE  "PIC7130 MODE 1=MAN 2=AUTO" %
%   N7:127  PIC7130_MAN_OP  "PIC7130 PY-7130 MANUAL OP (0-100%)" %
%   B3:38/0  "PY-7130 ALARM TRIGGERED OPEN STATE BIT" %
%   B3:42/12  "OSR" %
%   B16:4/2  PIC7130_AUTO_PB  "PIC7130 AUTO PUSHBUTTON ON HMI" %
%   N21:22/12  PIC7130_AUTO_DV  "PIC7130 AUTO MOMENTARY PB DeltaV -> PLC" %
%   B3:36/10  "OSR" %

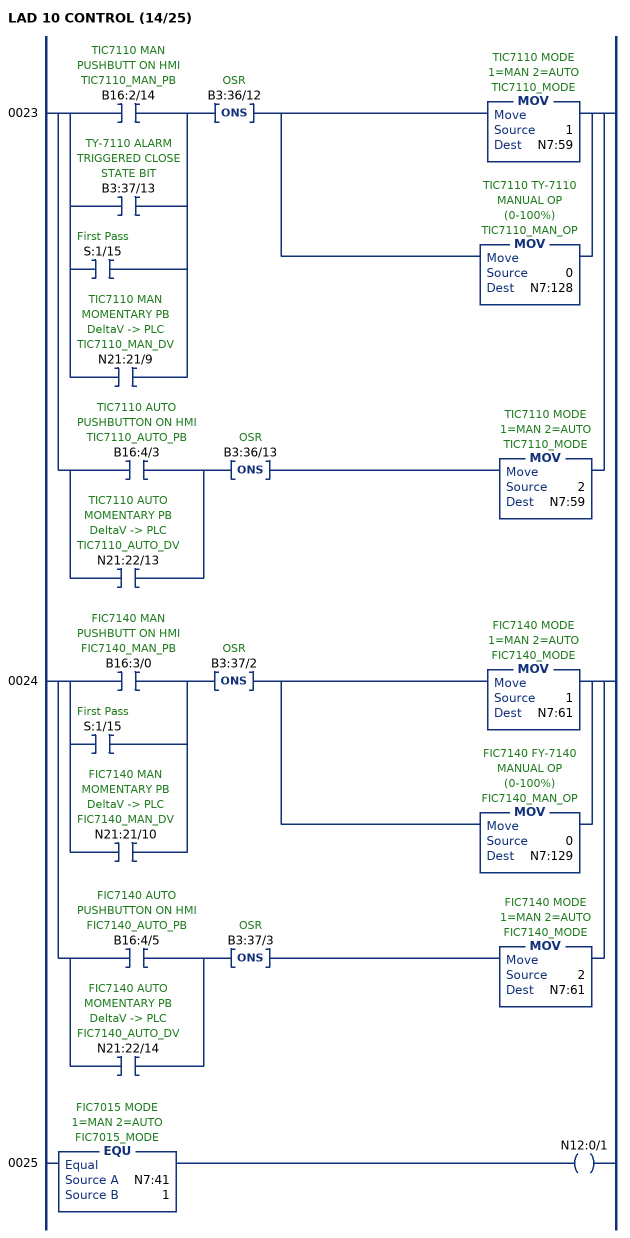
% Rung: 23 %
SOR BST BST XIC B16:2/14 NXB XIC B3:37/13 NXB XIC S:1/15 NXB XIC N21:21/9 BND OSR B3:36/12 BST MOV 1 N7:59 NXB MOV 0 N7:128 BND NXB BST XIC B16:4/3 NXB XIC N21:22/13 BND OSR B3:36/13 MOV 2 N7:59 BND EOR
%   B16:2/14  TIC7110_MAN_PB  "TIC7110 MAN PUSHBUTT ON HMI" %
%   B3:37/13  "TY-7110 ALARM TRIGGERED CLOSE STATE BIT" %
%   S:1/15  "First Pass" %
%   N21:21/9  TIC7110_MAN_DV  "TIC7110 MAN MOMENTARY PB DeltaV -> PLC" %
%   B3:36/12  "OSR" %
%   N7:59  TIC7110_MODE  "TIC7110 MODE 1=MAN 2=AUTO" %
%   N7:128  TIC7110_MAN_OP  "TIC7110 TY-7110 MANUAL OP (0-100%)" %
%   B16:4/3  TIC7110_AUTO_PB  "TIC7110 AUTO PUSHBUTTON ON HMI" %
%   N21:22/13  TIC7110_AUTO_DV  "TIC7110 AUTO MOMENTARY PB DeltaV -> PLC" %
%   B3:36/13  "OSR" %
% Rung: 24 %
SOR BST BST XIC B16:3/0 NXB XIC S:1/15 NXB XIC N21:21/10 BND OSR B3:37/2 BST MOV 1 N7:61 NXB MOV 0 N7:129 BND NXB BST XIC B16:4/5 NXB XIC N21:22/14 BND OSR B3:37/3 MOV 2 N7:61 BND EOR
%   B16:3/0  FIC7140_MAN_PB  "FIC7140 MAN PUSHBUTT ON HMI" %
%   S:1/15  "First Pass" %
%   N21:21/10  FIC7140_MAN_DV  "FIC7140 MAN MOMENTARY PB DeltaV -> PLC" %
%   B3:37/2  "OSR" %
%   N7:61  FIC7140_MODE  "FIC7140 MODE 1=MAN 2=AUTO" %
%   N7:129  FIC7140_MAN_OP  "FIC7140 FY-7140 MANUAL OP (0-100%)" %
%   B16:4/5  FIC7140_AUTO_PB  "FIC7140 AUTO PUSHBUTTON ON HMI" %
%   N21:22/14  FIC7140_AUTO_DV  "FIC7140 AUTO MOMENTARY PB DeltaV -> PLC" %
%   B3:37/3  "OSR" %
% Rung: 25 %
SOR EQU N7:41 1 OTE N12:0/1 EOR
%   N7:41  FIC7015_MODE  "FIC7015 MODE 1=MAN 2=AUTO" %

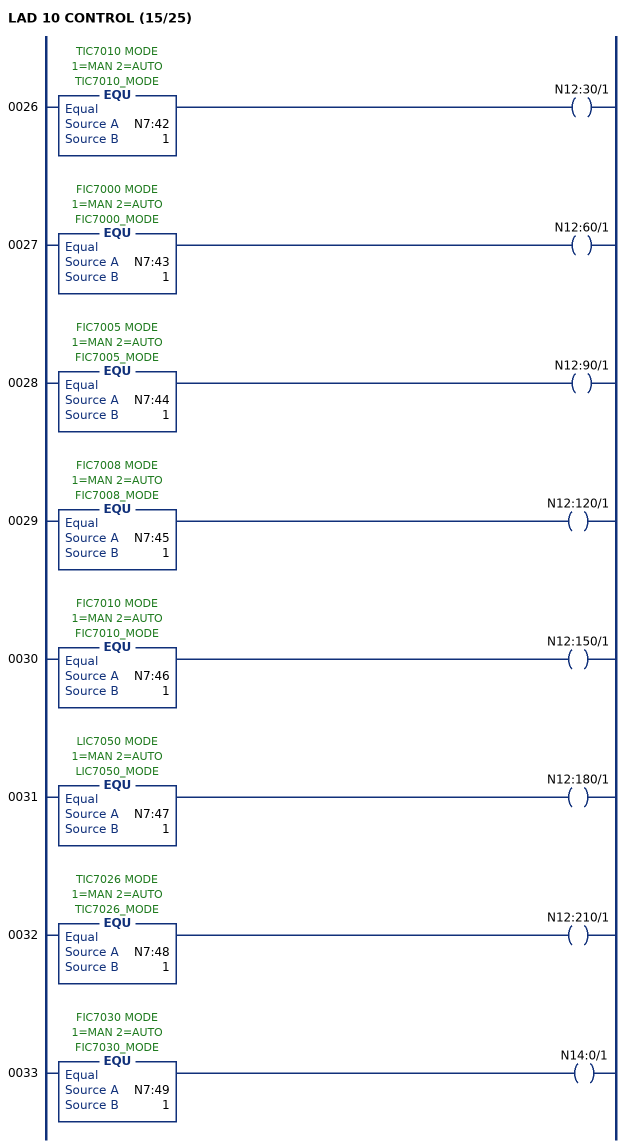
% Rung: 26 %
SOR EQU N7:42 1 OTE N12:30/1 EOR
%   N7:42  TIC7010_MODE  "TIC7010 MODE 1=MAN 2=AUTO" %
% Rung: 27 %
SOR EQU N7:43 1 OTE N12:60/1 EOR
%   N7:43  FIC7000_MODE  "FIC7000 MODE 1=MAN 2=AUTO" %
% Rung: 28 %
SOR EQU N7:44 1 OTE N12:90/1 EOR
%   N7:44  FIC7005_MODE  "FIC7005 MODE 1=MAN 2=AUTO" %
% Rung: 29 %
SOR EQU N7:45 1 OTE N12:120/1 EOR
%   N7:45  FIC7008_MODE  "FIC7008 MODE 1=MAN 2=AUTO" %
% Rung: 30 %
SOR EQU N7:46 1 OTE N12:150/1 EOR
%   N7:46  FIC7010_MODE  "FIC7010 MODE 1=MAN 2=AUTO" %
% Rung: 31 %
SOR EQU N7:47 1 OTE N12:180/1 EOR
%   N7:47  LIC7050_MODE  "LIC7050 MODE 1=MAN 2=AUTO" %
% Rung: 32 %
SOR EQU N7:48 1 OTE N12:210/1 EOR
%   N7:48  TIC7026_MODE  "TIC7026 MODE 1=MAN 2=AUTO" %
% Rung: 33 %
SOR EQU N7:49 1 OTE N14:0/1 EOR
%   N7:49  FIC7030_MODE  "FIC7030 MODE 1=MAN 2=AUTO" %

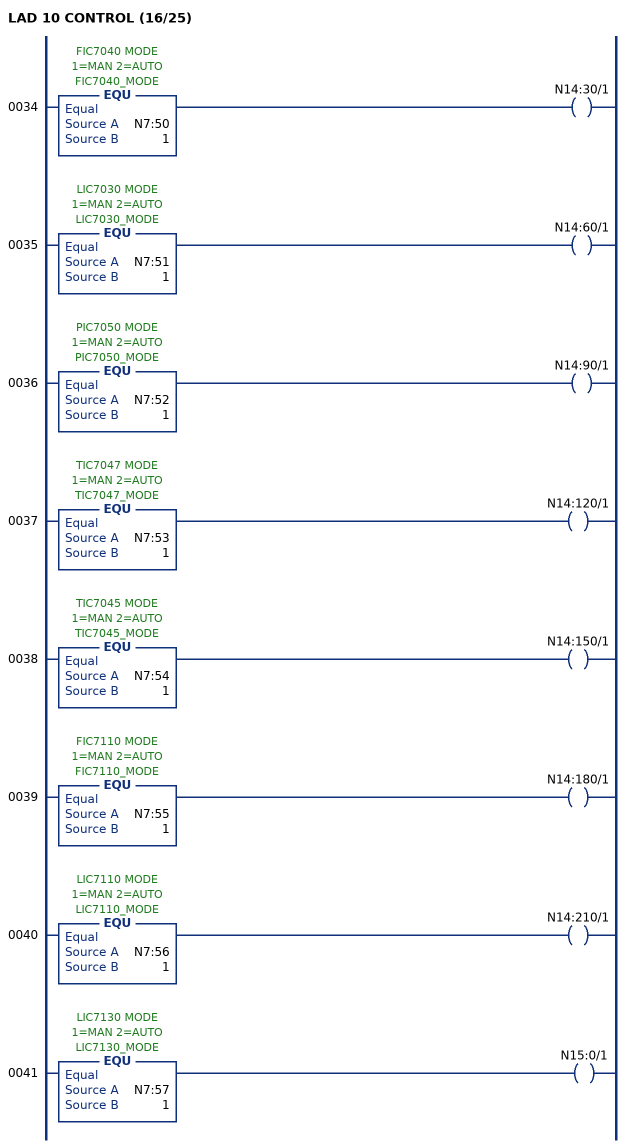
% Rung: 34 %
SOR EQU N7:50 1 OTE N14:30/1 EOR
%   N7:50  FIC7040_MODE  "FIC7040 MODE 1=MAN 2=AUTO" %
% Rung: 35 %
SOR EQU N7:51 1 OTE N14:60/1 EOR
%   N7:51  LIC7030_MODE  "LIC7030 MODE 1=MAN 2=AUTO" %
% Rung: 36 %
SOR EQU N7:52 1 OTE N14:90/1 EOR
%   N7:52  PIC7050_MODE  "PIC7050 MODE 1=MAN 2=AUTO" %
% Rung: 37 %
SOR EQU N7:53 1 OTE N14:120/1 EOR
%   N7:53  TIC7047_MODE  "TIC7047 MODE 1=MAN 2=AUTO" %
% Rung: 38 %
SOR EQU N7:54 1 OTE N14:150/1 EOR
%   N7:54  TIC7045_MODE  "TIC7045 MODE 1=MAN 2=AUTO" %
% Rung: 39 %
SOR EQU N7:55 1 OTE N14:180/1 EOR
%   N7:55  FIC7110_MODE  "FIC7110 MODE 1=MAN 2=AUTO" %
% Rung: 40 %
SOR EQU N7:56 1 OTE N14:210/1 EOR
%   N7:56  LIC7110_MODE  "LIC7110 MODE 1=MAN 2=AUTO" %
% Rung: 41 %
SOR EQU N7:57 1 OTE N15:0/1 EOR
%   N7:57  LIC7130_MODE  "LIC7130 MODE 1=MAN 2=AUTO" %

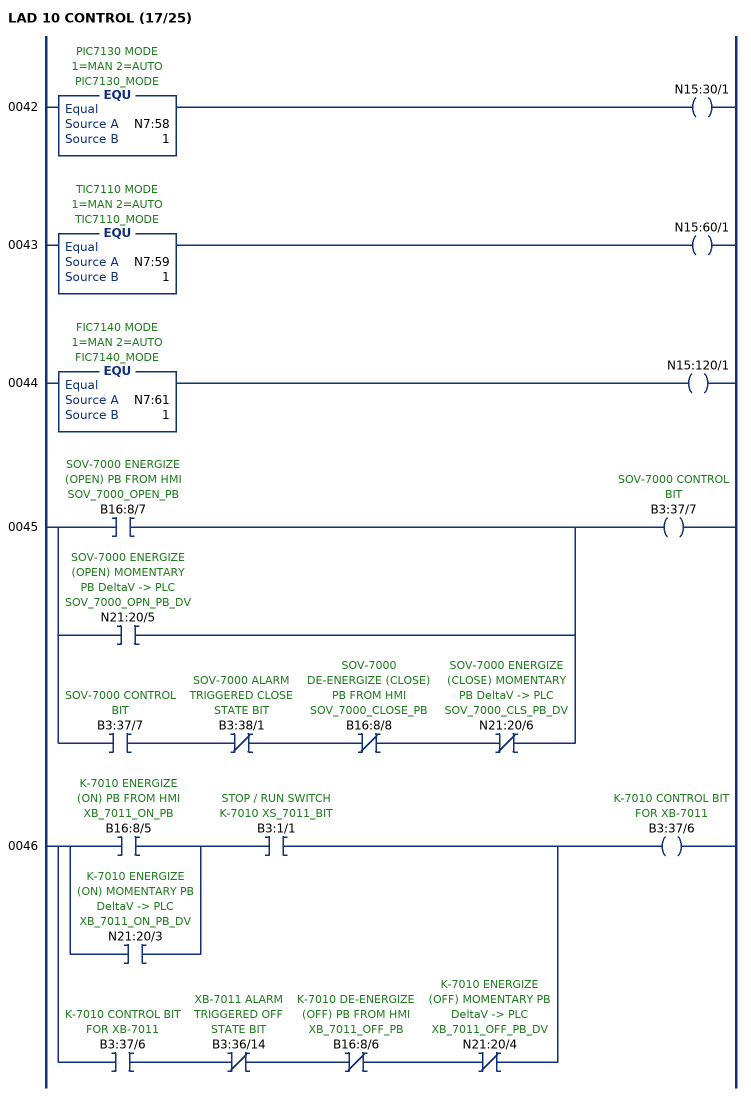
% Rung: 42 %
SOR EQU N7:58 1 OTE N15:30/1 EOR
%   N7:58  PIC7130_MODE  "PIC7130 MODE 1=MAN 2=AUTO" %
% Rung: 43 %
SOR EQU N7:59 1 OTE N15:60/1 EOR
%   N7:59  TIC7110_MODE  "TIC7110 MODE 1=MAN 2=AUTO" %
% Rung: 44 %
SOR EQU N7:61 1 OTE N15:120/1 EOR
%   N7:61  FIC7140_MODE  "FIC7140 MODE 1=MAN 2=AUTO" %
% Rung: 45 %
SOR BST BST XIC B16:8/7 NXB XIC N21:20/5 BND NXB XIC B3:37/7 XIO B3:38/1 XIO B16:8/8 XIO N21:20/6 BND OTE B3:37/7 EOR
%   B16:8/7  SOV_7000_OPEN_PB  "SOV-7000 ENERGIZE (OPEN) PB FROM HMI" %
%   N21:20/5  SOV_7000_OPN_PB_DV  "SOV-7000 ENERGIZE (OPEN) MOMENTARY PB DeltaV -> PLC" %
%   B3:37/7  "SOV-7000 CONTROL BIT" %
%   B3:38/1  "SOV-7000 ALARM TRIGGERED CLOSE STATE BIT" %
%   B16:8/8  SOV_7000_CLOSE_PB  "SOV-7000 DE-ENERGIZE (CLOSE) PB FROM HMI" %
%   N21:20/6  SOV_7000_CLS_PB_DV  "SOV-7000 ENERGIZE (CLOSE) MOMENTARY PB DeltaV -> PLC" %
% Rung: 46 %
SOR BST BST XIC B16:8/5 NXB XIC N21:20/3 BND XIC B3:1/1 NXB XIC B3:37/6 XIO B3:36/14 XIO B16:8/6 XIO N21:20/4 BND OTE B3:37/6 EOR
%   B16:8/5  XB_7011_ON_PB  "K-7010 ENERGIZE (ON) PB FROM HMI" %
%   N21:20/3  XB_7011_ON_PB_DV  "K-7010 ENERGIZE (ON) MOMENTARY PB DeltaV -> PLC" %
%   B3:1/1  XS_7011_BIT  "STOP / RUN SWITCH K-7010" %
%   B3:37/6  "K-7010 CONTROL BIT FOR XB-7011" %
%   B3:36/14  "XB-7011 ALARM TRIGGERED OFF STATE BIT" %
%   B16:8/6  XB_7011_OFF_PB  "K-7010 DE-ENERGIZE (OFF) PB FROM HMI" %
%   N21:20/4  XB_7011_OFF_PB_DV  "K-7010 ENERGIZE (OFF) MOMENTARY PB DeltaV -> PLC" %

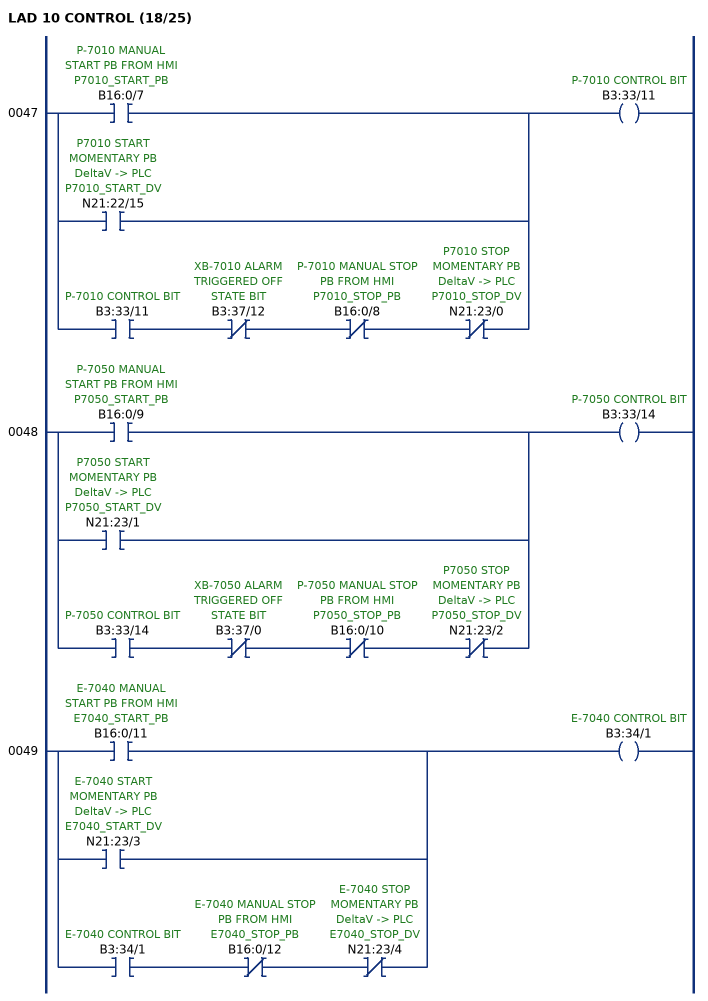
% Rung: 47 %
SOR BST BST XIC B16:0/7 NXB XIC N21:22/15 BND NXB XIC B3:33/11 XIO B3:37/12 XIO B16:0/8 XIO N21:23/0 BND OTE B3:33/11 EOR
%   B16:0/7  P7010_START_PB  "P-7010 MANUAL START PB FROM HMI" %
%   N21:22/15  P7010_START_DV  "P7010 START MOMENTARY PB DeltaV -> PLC" %
%   B3:33/11  "P-7010 CONTROL BIT" %
%   B3:37/12  "XB-7010 ALARM TRIGGERED OFF STATE BIT" %
%   B16:0/8  P7010_STOP_PB  "P-7010 MANUAL STOP PB FROM HMI" %
%   N21:23/0  P7010_STOP_DV  "P7010 STOP MOMENTARY PB DeltaV -> PLC" %
% Rung: 48 %
SOR BST BST XIC B16:0/9 NXB XIC N21:23/1 BND NXB XIC B3:33/14 XIO B3:37/0 XIO B16:0/10 XIO N21:23/2 BND OTE B3:33/14 EOR
%   B16:0/9  P7050_START_PB  "P-7050 MANUAL START PB FROM HMI" %
%   N21:23/1  P7050_START_DV  "P7050 START MOMENTARY PB DeltaV -> PLC" %
%   B3:33/14  "P-7050 CONTROL BIT" %
%   B3:37/0  "XB-7050 ALARM TRIGGERED OFF STATE BIT" %
%   B16:0/10  P7050_STOP_PB  "P-7050 MANUAL STOP PB FROM HMI" %
%   N21:23/2  P7050_STOP_DV  "P7050 STOP MOMENTARY PB DeltaV -> PLC" %
% Rung: 49 %
SOR BST BST XIC B16:0/11 NXB XIC N21:23/3 BND NXB XIC B3:34/1 XIO B16:0/12 XIO N21:23/4 BND OTE B3:34/1 EOR
%   B16:0/11  E7040_START_PB  "E-7040 MANUAL START PB FROM HMI" %
%   N21:23/3  E7040_START_DV  "E-7040 START MOMENTARY PB DeltaV -> PLC" %
%   B3:34/1  "E-7040 CONTROL BIT" %
%   B16:0/12  E7040_STOP_PB  "E-7040 MANUAL STOP PB FROM HMI" %
%   N21:23/4  E7040_STOP_DV  "E-7040 STOP MOMENTARY PB DeltaV -> PLC" %

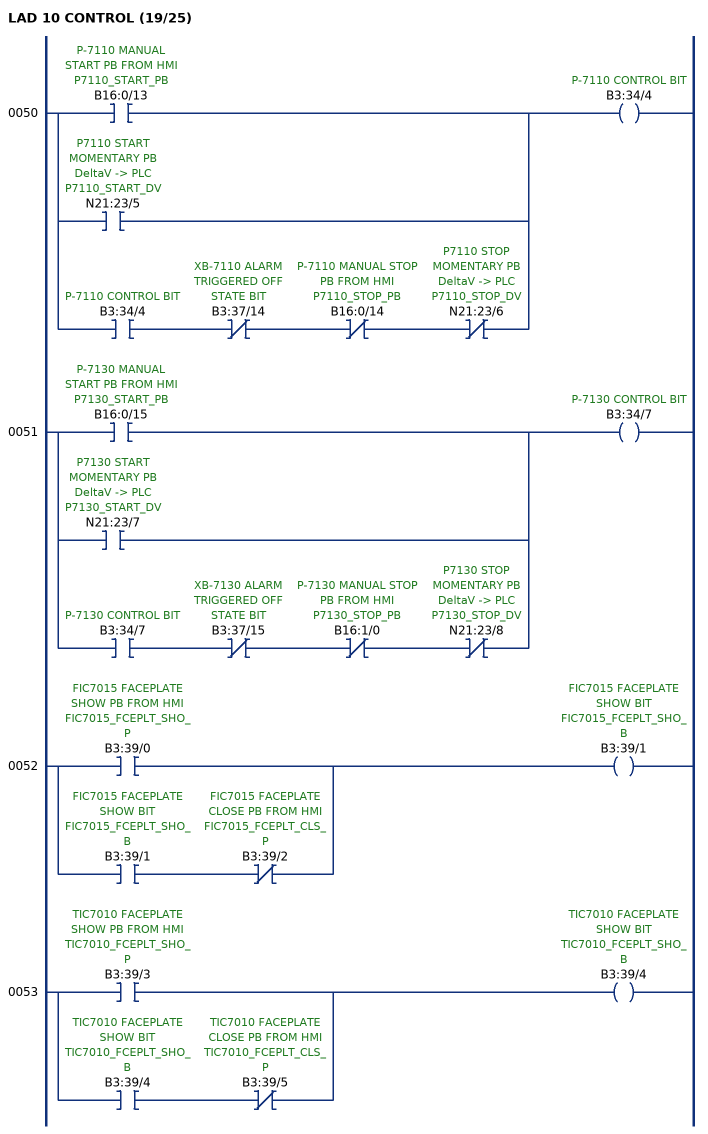
% Rung: 50 %
SOR BST BST XIC B16:0/13 NXB XIC N21:23/5 BND NXB XIC B3:34/4 XIO B3:37/14 XIO B16:0/14 XIO N21:23/6 BND OTE B3:34/4 EOR
%   B16:0/13  P7110_START_PB  "P-7110 MANUAL START PB FROM HMI" %
%   N21:23/5  P7110_START_DV  "P7110 START MOMENTARY PB DeltaV -> PLC" %
%   B3:34/4  "P-7110 CONTROL BIT" %
%   B3:37/14  "XB-7110 ALARM TRIGGERED OFF STATE BIT" %
%   B16:0/14  P7110_STOP_PB  "P-7110 MANUAL STOP PB FROM HMI" %
%   N21:23/6  P7110_STOP_DV  "P7110 STOP MOMENTARY PB DeltaV -> PLC" %
% Rung: 51 %
SOR BST BST XIC B16:0/15 NXB XIC N21:23/7 BND NXB XIC B3:34/7 XIO B3:37/15 XIO B16:1/0 XIO N21:23/8 BND OTE B3:34/7 EOR
%   B16:0/15  P7130_START_PB  "P-7130 MANUAL START PB FROM HMI" %
%   N21:23/7  P7130_START_DV  "P7130 START MOMENTARY PB DeltaV -> PLC" %
%   B3:34/7  "P-7130 CONTROL BIT" %
%   B3:37/15  "XB-7130 ALARM TRIGGERED OFF STATE BIT" %
%   B16:1/0  P7130_STOP_PB  "P-7130 MANUAL STOP PB FROM HMI" %
%   N21:23/8  P7130_STOP_DV  "P7130 STOP MOMENTARY PB DeltaV -> PLC" %
% Rung: 52 %
SOR BST XIC B3:39/0 NXB XIC B3:39/1 XIO B3:39/2 BND OTE B3:39/1 EOR
%   B3:39/0  FIC7015_FCEPLT_SHO_P  "FIC7015 FACEPLATE SHOW PB FROM HMI" %
%   B3:39/1  FIC7015_FCEPLT_SHO_B  "FIC7015 FACEPLATE SHOW BIT" %
%   B3:39/2  FIC7015_FCEPLT_CLS_P  "FIC7015 FACEPLATE CLOSE PB FROM HMI" %
% Rung: 53 %
SOR BST XIC B3:39/3 NXB XIC B3:39/4 XIO B3:39/5 BND OTE B3:39/4 EOR
%   B3:39/3  TIC7010_FCEPLT_SHO_P  "TIC7010 FACEPLATE SHOW PB FROM HMI" %
%   B3:39/4  TIC7010_FCEPLT_SHO_B  "TIC7010 FACEPLATE SHOW BIT" %
%   B3:39/5  TIC7010_FCEPLT_CLS_P  "TIC7010 FACEPLATE CLOSE PB FROM HMI" %

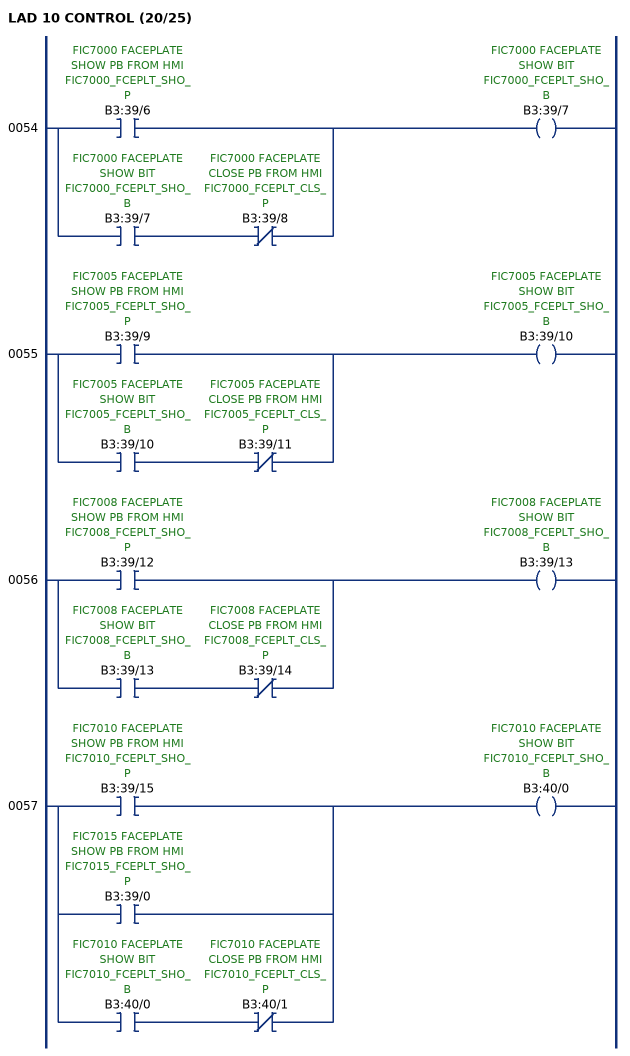
% Rung: 54 %
SOR BST XIC B3:39/6 NXB XIC B3:39/7 XIO B3:39/8 BND OTE B3:39/7 EOR
%   B3:39/6  FIC7000_FCEPLT_SHO_P  "FIC7000 FACEPLATE SHOW PB FROM HMI" %
%   B3:39/7  FIC7000_FCEPLT_SHO_B  "FIC7000 FACEPLATE SHOW BIT" %
%   B3:39/8  FIC7000_FCEPLT_CLS_P  "FIC7000 FACEPLATE CLOSE PB FROM HMI" %
% Rung: 55 %
SOR BST XIC B3:39/9 NXB XIC B3:39/10 XIO B3:39/11 BND OTE B3:39/10 EOR
%   B3:39/9  FIC7005_FCEPLT_SHO_P  "FIC7005 FACEPLATE SHOW PB FROM HMI" %
%   B3:39/10  FIC7005_FCEPLT_SHO_B  "FIC7005 FACEPLATE SHOW BIT" %
%   B3:39/11  FIC7005_FCEPLT_CLS_P  "FIC7005 FACEPLATE CLOSE PB FROM HMI" %
% Rung: 56 %
SOR BST XIC B3:39/12 NXB XIC B3:39/13 XIO B3:39/14 BND OTE B3:39/13 EOR
%   B3:39/12  FIC7008_FCEPLT_SHO_P  "FIC7008 FACEPLATE SHOW PB FROM HMI" %
%   B3:39/13  FIC7008_FCEPLT_SHO_B  "FIC7008 FACEPLATE SHOW BIT" %
%   B3:39/14  FIC7008_FCEPLT_CLS_P  "FIC7008 FACEPLATE CLOSE PB FROM HMI" %
% Rung: 57 %
SOR BST BST XIC B3:39/15 NXB XIC B3:39/0 BND NXB XIC B3:40/0 XIO B3:40/1 BND OTE B3:40/0 EOR
%   B3:39/15  FIC7010_FCEPLT_SHO_P  "FIC7010 FACEPLATE SHOW PB FROM HMI" %
%   B3:39/0  FIC7015_FCEPLT_SHO_P  "FIC7015 FACEPLATE SHOW PB FROM HMI" %
%   B3:40/0  FIC7010_FCEPLT_SHO_B  "FIC7010 FACEPLATE SHOW BIT" %
%   B3:40/1  FIC7010_FCEPLT_CLS_P  "FIC7010 FACEPLATE CLOSE PB FROM HMI" %

